RoboDK station: RobotStation.rdk

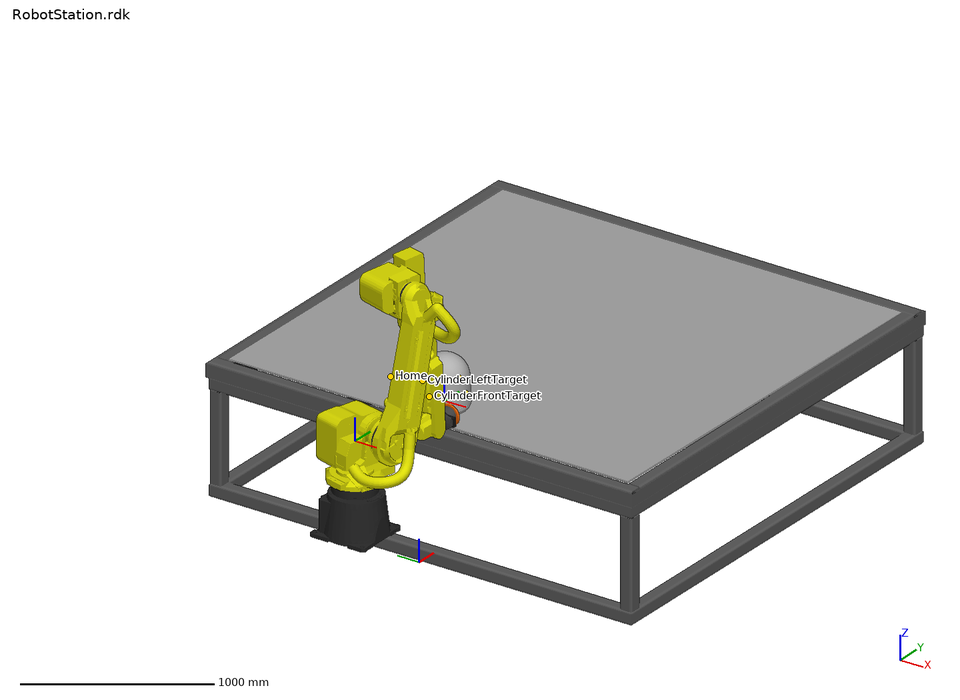
[picture v0: the station drawn from its stored meshes, robots at their saved joint values, targets as dots, program paths as lines]
Station RobotStation (saved by RoboDK 5.1.1). Poses are relative to the parent item; angles as X-Y-Z fixed-axis rotations.
  - frame Fanuc M-20iA/35M Base at (0, 0, 0) mm
    - robot Fanuc M-20iA/35M: 6 axes, payload 35 kg, reach 1813 mm, repeatability 0.04 mm, weight 252 kg
        modified DH rows (alpha deg, a mm, theta deg, d mm): 0, 0, 0, 525; -90, 150, -90, 0; 0, 790, 0, 0; -90, 150, 0, 860; 90, 0, 0, 0; -90, 0, 0, 100
        base shift (0, 0, -525) mm
        joint limits [-185, -110, -85, -200, -190, -450] to [185, 110, 245, 200, 190, 450]; home [0, 0, 0, 0, 0, 0]; saved at [75.264, 10.809, -87.104, -165.22, -85.199, -180.739]
      - tool RobotiQ Sanding Kit, TCP at (0, 0, 90.86) mm, size 127 x 139.7 x 103.3 mm
    - frame Frame 2 at (0, 800, -90) mm
      - object Radome at (0, 0, 0) mm, size 275.6 x 275.6 x 325.2 mm, geometry from FBB250 Antenna Radome.stl
      - target Home (Cartesian target) at (-201.49, -194.84, 158.53) mm, rotated rx -11.35 ry -84.72 rz -89.25 deg; joints [119.493, -11.647, -65.739, -41.293, 76.667, 14.757] of Fanuc M-20iA/35M
      - target CylinderFrontTarget (Cartesian target) at (0, -134, 78) mm, rotated rx 180 ry -88 rz 90 deg; joints [90, -2.65, -75.412, 0, 73.412, 0] of Fanuc M-20iA/35M
      - target CylinderLeftTarget (Cartesian target) at (-134, 0, 78) mm, rotated rx 180 ry -88 rz 0 deg; joints [112.094, 19.643, -69.031, 68.568, -95.851, -160.529] of Fanuc M-20iA/35M
      - target CylinderBackTarget (Cartesian target) at (0, 134, 78) mm, rotated rx 180 ry -88 rz -90 deg; joints [90, 32.139, -60.462, -180, 117.538, -360] of Fanuc M-20iA/35M
      - target CylinderRightTarget (Cartesian target) at (134, 0, 78) mm, rotated rx 180 ry -88 rz 180 deg; joints [67.906, 19.643, -69.031, -68.568, -95.851, -199.471] of Fanuc M-20iA/35M
    - frame Frame 3 at (0, 570, -922) mm, rotated rx 0 ry 0 rz 90 deg
      - object Table 108x114x32 IN at (0, 0, 0) mm, size 2628.9 x 2679.7 x 778.4 mm, geometry from Table-108x114x32-IN.sld
